ABB RobotStudio station: YuMi_Final_10-14-18.rspag

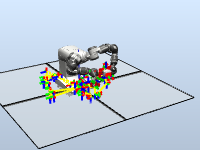
--- station ---
Station YuMi_Capstone_Final (saved by RobotStudio 6.7.7936.1011)
Controller Yumi_LF_Offline
  mechanical unit ROB_R: IRB14000_0.5_0.5_R, 6 joints, base frame (0, 0, 0) mm
  mechanical unit ROB_R_7: IRB14000_0.5_0.5_R, 1 joints, base frame (0, 0, 0) mm
  mechanical unit ROB_L: IRB14000_0.5_0.5_L, 6 joints, base frame (0, 0, 0) mm
  mechanical unit ROB_L_7: IRB14000_0.5_0.5_L, 1 joints, base frame (0, 0, 0) mm
Layout (positions relative to the parent item):
  - Smart_Gripper_Servo_One_Vacuum_Camera_Fingers [mechanism, from Tools\ABB_Smart_Gripper_Servo_One_Vacuum_Camera_Fingers.rslib] at (391.27, -12.04, 287.62) mm, rotated rx 179.56 ry 0.03 rz 94.75 deg; joint values [0.025] (rad or m)
  - Smart_Gripper_Servo_One_Vacuum_Camera_Fingers_2 [mechanism, from Tools\ABB_Smart_Gripper_Servo_One_Vacuum_Camera_Fingers.rslib] at (282.29, 267.76, 240.04) mm, rotated rx -93.42 ry -87.31 rz -179.37 deg; joint values [0.025] (rad or m)
  - IRB14000_0.5_0.5_2 [mechanism, from Robots\IRB14000_0.5_0.5__01.rslib] at (0, 0, 0) mm
  - IRB14000_0.5_0.5_R [mechanism, from Robots\IRB14000_0.5_0.5__01.rslib] at (0, 0, 0) mm; joint values [1.4938, -0.7266, -1.3651, 0.7569, 4.3395, 1.3243, -3.2623] (rad or m)
  - IRB14000_0.5_0.5_L [mechanism, from Robots\IRB14000_0.5_0.5__01.rslib] at (0, 0, 0) mm; joint values [-0.6453, -1.1889, 1.5214, 0.5648, 0.0097, 1.2191, -0.4517] (rad or m)
Attachment: Smart_Gripper_Servo_One_Vacuum_Camera_Fingers is attached to IRB14000_0.5_0.5_R / Link7
Attachment: Smart_Gripper_Servo_One_Vacuum_Camera_Fingers_2 is attached to IRB14000_0.5_0.5_L / Link7
Targets, tools, work objects and paths stored in the station and not in the controller backup, written as RAPID:
! task T_ROB_R
MODULE MainModule
  VAR syncident sync1;
  VAR syncident sync2;
  VAR syncident sync3;
  VAR syncident sync4;
  VAR syncident sync5;
  VAR syncident sync6;
  VAR syncident sync7;
  VAR syncident sync8;
  VAR syncident sync9;
  VAR syncident sync10;
  VAR syncident sync11;
  VAR syncident sync12;
  VAR syncident sync13;
  VAR syncident sync14;
  VAR syncident sync15;
  VAR syncident sync16;
  VAR syncident sync17;
ENDMODULE

! task T_ROB_R
MODULE CalibData
  PERS tooldata Servo:=[TRUE,[[0,0,114.2],[1,0,0,0]],[0.24,[8.2,12.5,48.1],[1,0,0,0],0.00022,0.00024,0.00009]];
  PERS tooldata VaccumOne:=[TRUE,[[56,18.5,37.5],[0.707106781,0,0.707106781,0]],[0.24,[8.2,12.5,48.1],[1,0,0,0],0.00022,0.00024,0.00009]];
  PERS tooldata Camera:=[TRUE,[[-7.3,28.3,35.1],[0.5,-0.5,0.5,0.5]],[0.24,[8.2,12.5,48.1],[1,0,0,0],0.00022,0.00024,0.00009]];
ENDMODULE

! task T_ROB_L
MODULE MainModule
  VAR syncident sync1;
  VAR syncident sync2;
  VAR syncident sync3;
  VAR syncident sync4;
  VAR syncident sync5;
  VAR syncident sync6;
  VAR syncident sync7;
  VAR syncident sync8;
  VAR syncident sync9;
  VAR syncident sync10;
  VAR syncident sync11;
  VAR syncident sync12;
  VAR syncident sync13;
  VAR syncident sync14;
  VAR syncident sync15;
  VAR syncident sync16;
  VAR syncident sync17;
ENDMODULE

! task T_ROB_L
MODULE CalibData
  PERS tooldata Servo:=[TRUE,[[0,0,114.2],[1,0,0,0]],[0.24,[8.2,12.5,48.1],[1,0,0,0],0.00022,0.00024,0.00009]];
  PERS tooldata VaccumOne:=[TRUE,[[56,18.5,37.5],[0.707106781,0,0.707106781,0]],[0.24,[8.2,12.5,48.1],[1,0,0,0],0.00022,0.00024,0.00009]];
  PERS tooldata Camera:=[TRUE,[[-7.3,28.3,35.1],[0.5,-0.5,0.5,0.5]],[0.24,[8.2,12.5,48.1],[1,0,0,0],0.00022,0.00024,0.00009]];
ENDMODULE

! task T_ROB_R
MODULE CalibData
  PERS tooldata Servo:=[TRUE,[[0,0,114.2],[1,0,0,0]],[0.24,[8.2,12.5,48.1],[1,0,0,0],0.00022,0.00024,0.00009]];
  PERS tooldata VaccumOne:=[TRUE,[[56,18.5,37.5],[0.707106781,0,0.707106781,0]],[0.24,[8.2,12.5,48.1],[1,0,0,0],0.00022,0.00024,0.00009]];
  PERS tooldata Camera:=[TRUE,[[-7.3,28.3,35.1],[0.5,-0.5,0.5,0.5]],[0.24,[8.2,12.5,48.1],[1,0,0,0],0.00022,0.00024,0.00009]];
ENDMODULE

! task T_ROB_L
MODULE CalibData
  PERS tooldata Servo:=[TRUE,[[0,0,114.2],[1,0,0,0]],[0.24,[8.2,12.5,48.1],[1,0,0,0],0.00022,0.00024,0.00009]];
  PERS tooldata VaccumOne:=[TRUE,[[56,18.5,37.5],[0.707106781,0,0.707106781,0]],[0.24,[8.2,12.5,48.1],[1,0,0,0],0.00022,0.00024,0.00009]];
  PERS tooldata Camera:=[TRUE,[[-7.3,28.3,35.1],[0.5,-0.5,0.5,0.5]],[0.24,[8.2,12.5,48.1],[1,0,0,0],0.00022,0.00024,0.00009]];
ENDMODULE


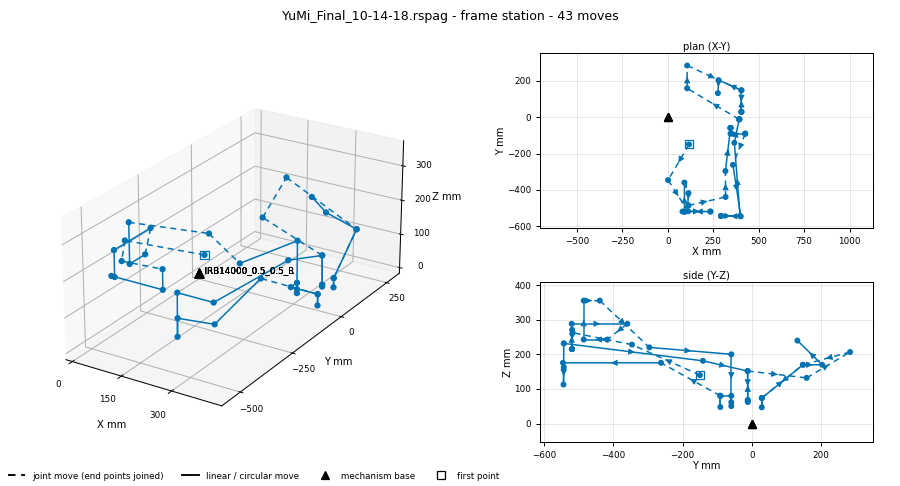
[picture p0: tool path of YuMi_Final_10-14-18.rspag in frame station, 43 of 43 moves have a stored position in this frame; points joined in program order, loops and branches not executed]
--- Backups/Yumi_LF_Offline/RAPID/TASK1/PROGMOD/MainModule.mod ---
MODULE MainModule
    !******************************************************************
    !* Station : YuMi Work Cell
    !******************************************************************
    !* Customer : McMaster University
    !* Project Name : Electronic Screwdriver Assembly
    !*
    !* Robot Model : IRB 14000
    !* Software : RobotWare 6.07
    !*
    !* Authors : Simran Nijjar, Justin Grimm, Samony Riyaz, Amy Hasselman
    !* Company : McMaster University
    !* City/Province : Hamilton, Ontario
    !* Department : W. Booth School of Engineering Practice & Technology
    !* Telephone : N/A
    !*
    !* Program: T_ROB_R
    !* Created : 2018-09-18
    !* Version : 1.0
    !*
    !******************************************************************

    !General Declaration
    PERS tasks task_list{2} := [ ["T_ROB_R"], ["T_ROB_L"] ];
    VAR syncident sync1; !Sync Arm Home Positions
    VAR syncident sync2; !Sync Gripper Open Position
    VAR syncident sync3; !Sync Gripper Close Position
    VAR syncident sync4; !Sync GrommetBin Position1
    VAR syncident sync5; !Sync GrommetBin Position2
    VAR syncident sync6; !Sync GrommetBin Position3
    VAR syncident sync7; !Sync GrommetBin Position4

    !Communication Declaration
    VAR socketdev server;
    VAR socketdev client;
    VAR string message;
    VAR rawbytes data;


	PROC main()
        !Move to Home Position
		MoveJ [[116.737861724,-149.931251033,139.878323961],[0.062653888,-0.842399836,-0.108469979,-0.524090898],[0,0,0,4],[-101.221,9E+09,9E+09,9E+09,9E+09,9E+09]], v1000, z50, tGripper;
		!MoveJ [[110.29,-313.83,302.97],[0.320874,0.00713782,0.947055,0.00865406],[0,1,2,5],[-110.474,9E+09,9E+09,9E+09,9E+09,9E+09]], v1000, z50, tool0;
        WaitSyncTask \InPos, sync1, task_list \TimeOut := 60;

        !Calibrate Grippers
        GripperInitialization;

        !Grippers Initialized Comformation
        g_MoveTo 0;
        WaitRob \InPos;
        WaitSyncTask \InPos, sync2, task_list \TimeOut := 60;

        g_MoveTo 15;
        WaitRob \InPos;
        WaitSyncTask \InPos, sync3, task_list \TimeOut := 60;

        !Move Screwdriver Bin to Correct Position
        MoveJ [[1.625300521,-346.188591473,227.922111416],[0.007707619,0.999903927,-0.000742016,0.011496899],[0,-1,1,4],[-70.2983,9E+09,9E+09,9E+09,9E+09,9E+09]], v1000, z50, tGripper;
        MoveJ [[111.921573894,-517.679338441,262.371959938],[0.007636972,0.999904216,-0.000728005,0.011519802],[0,-1,2,4],[-72.7464,9E+09,9E+09,9E+09,9E+09,9E+09]], v1000, z50, tGripper;
        MoveJ [[234.314486144,-519.240905612,270.651668137],[0.007608269,0.999904877,-0.0005289,0.011492199],[0,-1,2,4],[-162.822,9E+09,9E+09,9E+09,9E+09,9E+09]], v1000, z50, tGripper;
        g_MoveTo 0;
        WaitRob \InPos;
        MoveL [[234.312932861,-519.240747252,215.101630035],[0.00760767,0.999904947,-0.000530615,0.011486499],[0,-1,2,4],[-162.825,9E+09,9E+09,9E+09,9E+09,9E+09]], v1000, z50, tGripper;
        MoveL [[80.782123738,-519.239699323,215.101595493],[0.00760385,0.999905012,-0.00052779,0.0114835],[0,0,1,4],[-162.828,9E+09,9E+09,9E+09,9E+09,9E+09]], v100, z50, tGripper;
        MoveL [[91.392040059,-520.360093654,215.101599575],[0.00760529,0.999905004,-0.000528675,0.0114832],[0,0,1,4],[-162.831,9E+09,9E+09,9E+09,9E+09,9E+09]], v200, z50, tGripper;
        MoveL [[91.399265315,-520.341509224,288.241945811],[0.007536403,0.999904343,-0.000572503,0.011583604],[0,-1,1,4],[-46.5055,9E+09,9E+09,9E+09,9E+09,9E+09]], v200, z50, tGripper;
        WaitRob \InPos;
        MoveL [[91.398688306,-359.668522139,288.241887402],[0.007525373,0.999904448,-0.00057653,0.011581505],[0,-1,2,4],[-46.5056,9E+09,9E+09,9E+09,9E+09,9E+09]], v200, z50, tGripper;
        WaitRob \InPos;
        MoveJ [[113.281646346,-417.364249351,242.672999782],[0.496441086,0.502834087,-0.499757087,0.500946087],[0,1,-1,4],[-119.673,9E+09,9E+09,9E+09,9E+09,9E+09]], v200, z50, tGripper;

        g_MoveTo 9;
        WaitRob \InPos;
        MoveL [[113.281646863,-485.724250766,242.673272807],[0.496441087,0.502833088,-0.499757088,0.500947088],[0,1,0,4],[-119.673,9E+09,9E+09,9E+09,9E+09,9E+09]], v200, z50, tGripper;
        WaitRob \InPos;
        g_GripIn \holdForce :=12;
        MoveL [[113.282188675,-485.724252296,355.154359115],[0.496443089,0.502833091,-0.49975309,0.50094909],[0,2,0,4],[-119.675,9E+09,9E+09,9E+09,9E+09,9E+09]], v200, z50, tGripper;
        MoveJ [[317.912323563,-439.194244895,355.153131276],[0.496442332,0.502837336,-0.499753334,0.500945335],[1,1,-1,4],[-119.678,9E+09,9E+09,9E+09,9E+09,9E+09]], v200, z50, tGripper;
        MoveJ [[317.022439031,-296.105779981,220.044708012],[0.0188621,-0.709563985,0.704158986,0.0179804],[1,3,-1,4],[-119.677,9E+09,9E+09,9E+09,9E+09,9E+09]], v200, z50, tGripper;
        MoveL [[344.96,-59.21,200.05],[0.00733667,-0.709769,0.704368,0.00639342],[1,3,0,4],[157.039,9E+09,9E+09,9E+09,9E+09,9E+09]], v200, z50, tGripper;
        WaitSyncTask \InPos, sync4, task_list \TimeOut := 60;
        MoveL [[344.96,-59.21,61.37],[0.00734294,-0.709766,0.70437,0.00639399],[1,3,0,4],[157.041,9E+09,9E+09,9E+09,9E+09,9E+09]], v20, z50, tGripper;
        MoveL [[344.96,-59.21,50.36],[0.00734279,-0.709765,0.704371,0.00639592],[1,3,0,4],[157.039,9E+09,9E+09,9E+09,9E+09,9E+09]], v20, z50, tGripper;
        WaitRob \InPos;
        g_MoveTo 6;
        WaitRob \InPos;
        WaitSyncTask \InPos, sync5, task_list \TimeOut := 60;
        WaitSyncTask \InPos, sync6, task_list \TimeOut := 60;
        MoveL [[344.95,-59.21,80.07],[0.0073388,-0.709769,0.704367,0.00639981],[1,3,0,4],[157.039,9E+09,9E+09,9E+09,9E+09,9E+09]], v20, z50, tGripper;
        MoveL [[344.95,-90.89,80.07],[0.00733899,-0.70977,0.704366,0.00640178],[1,3,0,4],[157.038,9E+09,9E+09,9E+09,9E+09,9E+09]], v20, z50, tGripper;
        WaitSyncTask \InPos, sync7, task_list \TimeOut := 60;
        MoveL [[425.74,-90.89,80.07],[0.00733914,-0.709769,0.704367,0.00640155],[1,3,0,4],[157.038,9E+09,9E+09,9E+09,9E+09,9E+09]], v20, z50, tGripper;
        MoveL [[425.74,-90.89,47.66],[0.00734079,-0.709768,0.704368,0.00640208],[1,3,0,4],[157.038,9E+09,9E+09,9E+09,9E+09,9E+09]], v20, z50, tGripper;
        WaitRob \InPos;
        g_MoveTo 12;
        WaitRob \InPos;
        MoveL [[425.74,-90.89,80.07],[0.00733914,-0.709769,0.704367,0.00640155],[1,3,0,4],[157.038,9E+09,9E+09,9E+09,9E+09,9E+09]], v20, z50, tGripper;
        MoveJ [[358.12,-262.41,175.42],[0.00734778,-0.709763,0.704373,0.00641492],[0,3,-1,4],[157.036,9E+09,9E+09,9E+09,9E+09,9E+09]], v200, z50, tGripper;
        MoveL [[401.48,-545.66,175.40],[0.00980935,-0.999797,0.0175768,-0.000449508],[1,3,-2,4],[-152.759,9E+09,9E+09,9E+09,9E+09,9E+09]], v200, z50, tGripper;
        MoveL [[292.66,-543.24,162.68],[0.00981674,-0.999797,0.0175764,-0.000446634],[0,3,-2,4],[-152.763,9E+09,9E+09,9E+09,9E+09,9E+09]], v20, z50, tGripper;
        MoveL [[292.39,-544.14,112.56],[0.00982093,-0.999936,-0.00555262,-0.000675012],[0,3,-2,4],[-152.771,9E+09,9E+09,9E+09,9E+09,9E+09]], v20, z50, tGripper;
        WaitRob \InPos;
        g_MoveTo 6;
        WaitRob \InPos;
        g_GripIn \holdForce := 12;
        WaitRob \InPos;
        MoveL [[292.66,-543.25,231.50],[0.00981188,-0.999797,0.0175706,-0.000448127],[0,3,-2,4],[-152.762,9E+09,9E+09,9E+09,9E+09,9E+09]], v20, z50, tGripper;
        MoveL [[397.32,-543.24,231.50],[0.00980798,-0.999797,0.0175712,-0.000449308],[1,3,-2,4],[-152.763,9E+09,9E+09,9E+09,9E+09,9E+09]], v20, z50, tGripper;
        MoveL [[366.17,-140.98,181.13],[0.00267605,0.705528,0.708672,0.00274474],[1,3,-2,4],[166.603,9E+09,9E+09,9E+09,9E+09,9E+09]], v200, z50, tGripper;
        MoveL [[392.31,-12.03,151.62],[0.00277692,0.677184,0.735803,0.00262845],[1,3,-2,4],[166.306,9E+09,9E+09,9E+09,9E+09,9E+09]], v200, z50, tGripper;
        MoveL [[393.44,-11.60,67.62],[0.00277557,0.677187,0.735801,0.0026324],[1,3,-2,4],[166.306,9E+09,9E+09,9E+09,9E+09,9E+09]], v20, z50, tGripper;
        MoveL [[393.44,-11.60,62.17],[0.00277571,0.677187,0.735801,0.00263129],[1,3,-2,4],[166.306,9E+09,9E+09,9E+09,9E+09,9E+09]], v10, z50, tGripper;
        WaitRob \InPos;
        g_MoveTo 12;
        WaitRob \InPos;
        MoveL [[393.44,-11.60,67.62],[0.00277557,0.677187,0.735801,0.0026324],[1,3,-2,4],[166.306,9E+09,9E+09,9E+09,9E+09,9E+09]], v20, z50, tGripper;
        MoveL [[392.31,-12.03,151.62],[0.00277692,0.677184,0.735803,0.00262845],[1,3,-2,4],[166.306,9E+09,9E+09,9E+09,9E+09,9E+09]], v200, z50, tGripper;













!        !Create communication
!        SocketCreate server;
!        SocketBind server, "10.0.13.12", 55000;
!        SocketListen server;
!        SocketAccept server, client;

!        !Send message to the client
!        !SocketSend client\Str:="Hello me!";

!        FOR i FROM 1 TO 10 DO
!            SocketSend client\Str:="Hello me!";
!        ENDFOR


!        !Receive a message from the client
!        SocketReceive client, \RawData:=data;
!        UnpackRawBytes data,1,message\ASCII:=15;

!        !Close communication
!        SocketClose server;


    ENDPROC




    PROC GripperInitialization()
            !Initialization code
            VAR num GripperState;
            VAR bool GripperCalibrated;

            !Check gripper is powered on and calibrated
            GripperState:=g_GetState();
            TPWrite ": Gripper State: "\Num:=GripperState;
            GripperCalibrated:=g_IsCalibrated();

            IF (Not GripperCalibrated) THEN
                g_Init\Calibrate;
            ENDIF

            RETURN;

        ERROR
            IF (ERRNO=ERR_NORUNUNIT) THEN TPWrite " Gripper not powered on.";
                EXIT;
            ENDIF
            TPWrite " Init. - Unhandled Error. #"\Num:=ERRNO;
            EXIT;
    ENDPROC





ENDMODULE

--- Backups/Yumi_LF_Offline/RAPID/TASK1/SYSMOD/LINKEDM.sys ---
%%%
  VERSION:1
  LANGUAGE:ENGLISH
%%%

MODULE LINKEDM (SYSMODULE)

! FOLLOWER
!     Name of electronically linked follower axis used by operator at teach pendent.
      PERS string l_f_axis_name{5}       :=  ["",  "", "", "", ""];

!     Name of the mechanical unit for follower axis.
      PERS string l_f_mecunt_n{5}  :=  ["", "", "", "", ""];

!     Linked follower axis number in the mechanical unit (first axis in mech. unit is number 1).
      PERS num l_f_axis_no{5}      :=  [0,          0,   0,  0,  0];

! MASTER
!     Name of the mechanical unit for linked master axis.
      PERS string l_m_mecunt_n{5} :=  ["", "", "", "", ""];

!     Linked master axis number in the mechanical unit (first axis in mech. unit is number 1).
!     See axis number table in documentation for different master mechanical units.
      PERS num l_m_axis_no{5}     :=  [0,  0,  0,  0,  0];

! POSITION OFFSET
!     The increase of the allowed offset position between the master and follower
!     positions, used when starting AUTO mode. As soon as the offset is decreased
!     the old configurated parameter is used.
!     Example: 3 => the configurated value of allowed offset is increased 3 times.
      PERS num offset_ratio{5}       :=  [10,  10,   10,  10,  10];

! SPEED RATIO
!     Speed_ratio used in AUTO and JOG modes [ very_slow   slow    normal    fast]
!     Value 1 = max allowed manual speed.
      CONST num speed_ratio {20}      := [0.01, 0.01, 0.01, 0.01, 0.01,
                                          0.05, 0.05, 0.05, 0.05, 0.05,
                                          0.20, 0.20, 0.20, 0.20, 0.20,
                                          1.00, 1.00, 1.00, 1.00, 1.00];

! STEP SIZE
!     Displacement position used in JOG mode for each activation of positive or
!     negative movement.                  [very_short    short   normal   long]
!     Unit degees or meter.
      CONST num displacement {20}     := [0.001, 0.001, 0.001, 0.001, 0.001,
                                          0.005, 0.005, 0.005, 0.005, 0.005,
                                          0.020, 0.020, 0.020, 0.020, 0.020,
                                          0.100, 0.100, 0.100, 0.100, 0.100];


!-------------------------------------------------------------
 PROC Linked_m ()
      Linked_m_exe ;
 ENDPROC
ENDMODULE

--- Backups/Yumi_LF_Offline/RAPID/TASK1/SYSMOD/YuMiLib_Params_R.sys ---
MODULE YuMiLib_Params_R(SYSMODULE)
    !***************************************************************************
    !*                              Common parameters                          *
    !***************************************************************************
    CONST loaddata ld_YuMiGripper_S:=[0.230,[8.2,11.7,52.0],[1,0,0,0],0.00021,0.00024,0.00009];
    CONST loaddata ld_YuMiGripper_S_V1:=[0.248,[8.6,11.7,52.7],[1,0,0,0],0.00021,0.00024,0.00009];
    CONST loaddata ld_YuMiGripper_S_V1_V2:=[0.280,[7.1,11.9,47.3],[1,0,0,0],0.00025,0.00029,0.00012];
    CONST loaddata ld_YuMiGripper_S_C:=[0.244,[7.5,11.8,52.7],[1,0,0,0],0.00021,0.00023,0.00008];
    CONST loaddata ld_YuMiGripper_S_C_V1:=[0.262,[7.8,11.9,50.7],[1,0,0,0],0.00022,0.00024,0.00009];

    !***************************************************************************
    ! Predefined tools for different configurations of the Standard Smart Gripper
    !***************************************************************************
    TASK PERS tooldata tHandCamera:=[TRUE,[[-7.79332,26.2553,35.637],[0.507106,-0.492819,-0.512337,-0.487323]],[0.262,[7.8,11.9,50.7],[1,0,0,0],0.00022,0.00024,0.00009]];
    TASK PERS tooldata tGripper:=[TRUE,[[0,0,136],[1,0,0,0]],[0.23,[8.2,11.7,52],[1,0,0,0],0.00021,0.00024,0.00009]];
    TASK PERS tooldata tVacuum1:=[TRUE,[[63.5,18.5,37.5],[0.707106781,0,0.707106781,0]],[0.248,[8.6,11.7,52.7],[1,0,0,0],0.00021,0.00024,0.00009]];
    TASK PERS tooldata tVacuum2:=[TRUE,[[-63.5,18.5,37.5],[0.707106781,0,-0.707106781,0]],[0.28,[7.1,11.9,47.3],[1,0,0,0],0.00025,0.00029,0.00012]];

    !***************************************************************************
    !*                         Task specific paramters                         *
    !***************************************************************************

    TASK PERS wobjdata WObj_FollowRobL:=[FALSE,FALSE,"ROB_L",[[0,0,0],[1,0,0,0]],[[0,0,0],[1,0,0,0]]];
    TASK PERS wobjdata WObj_Vision:=[FALSE,TRUE,"",[[401.591,32.4092,0],[0.424655,-0.000000122,-0.000000191,0.905355]],[[0,0,0],[1,0,0,0]]];

    !**************************************************************************
    !*                                Speeddata                               *
    !**************************************************************************
    CONST speeddata vSlow:=[100,50,5000,1000];
    CONST speeddata vMedium:=[300,150,5000,1000];
    CONST speeddata vFast:=v1000;

ENDMODULE

--- Backups/Yumi_LF_Offline/RAPID/TASK2/PROGMOD/MainModule.mod ---
MODULE MainModule
    !******************************************************************
    !* Station : YuMi Work Cell
    !******************************************************************
    !* Customer : McMaster University
    !* Project Name : Electronic Screwdriver Assembly
    !*
    !* Robot Model : IRB 14000
    !* Software : RobotWare 6.07
    !*
    !* Authors : Simran Nijjar, Justin Grimm, Samony Riyaz, Amy Hasselman
    !* Company : McMaster University
    !* City/Province : Hamilton, Ontario
    !* Department : W. Booth School of Engineering Practice & Technology
    !* Telephone : N/A
    !*
    !* Program: T_ROB_L
    !* Created : 2018-09-18
    !* Version : 1.0
    !*
    !******************************************************************

    !General Declaration
    PERS tasks task_list{2} := [ ["T_ROB_R"], ["T_ROB_L"] ];
    VAR syncident sync1; !Sync Arm Home Positions
    VAR syncident sync2; !Sync Gripper Open Position
    VAR syncident sync3; !Sync Gripper Close Position
    VAR syncident sync4; !Sync GrommetBin Position1
    VAR syncident sync5; !Sync GrommetBin Position2
    VAR syncident sync6; !Sync GrommetBin Position3
    VAR syncident sync7; !Sync GrommetBin Position4

    !Communication Declaration
    VAR socketdev server;
    VAR socketdev client;
    VAR string message;
    VAR rawbytes data;


    PROC main()
		MoveJ [[106.445211471,158.554553337,131.92293514],[0.04782649,0.851736822,-0.124160974,0.506794894],[0,0,0,4],[101.293,9E+09,9E+09,9E+09,9E+09,9E+09]], v1000, z50, tGripper;
		!MoveJ [[97.79,299.03,304.48],[0.0114881,-0.942459,0.0541276,-0.329712],[0,-2,-2,4],[108.747,9E+09,9E+09,9E+09,9E+09,9E+09]], v1000, z50, tool0;
        WaitSyncTask \InPos, sync1, task_list \TimeOut := 60;

        !Calibrate Grippers
        GripperInitialization;

        !Grippers Initialized Comformation
        g_MoveTo 0;
        WaitRob \InPos;
        WaitSyncTask \InPos, sync2, task_list \TimeOut := 60;

        g_MoveTo 15;
        WaitRob \InPos;
        WaitSyncTask \InPos, sync3, task_list \TimeOut := 60;

        !Remove Grommet from Right Screwdriver Shell
        WaitSyncTask \InPos, sync4, task_list \TimeOut := 60;
        MoveJ [[106.46,283.94,206.53],[0.0478122,0.85173,-0.124169,0.506805],[0,0,0,4],[101.295,9E+09,9E+09,9E+09,9E+09,9E+09]], v200, z50, tGripper;
        MoveJ [[404.90,147.80,169.77],[0.009872,-0.723527,-0.690004,0.0174687],[-1,1,0,4],[-169.944,9E+09,9E+09,9E+09,9E+09,9E+09]], v200, z50, tGripper;
        WaitSyncTask \InPos, sync5, task_list \TimeOut := 60;
        MoveL [[404.90,28.94,73.67],[0.0098782,-0.723515,-0.690017,0.0174677],[-1,2,0,4],[146.542,9E+09,9E+09,9E+09,9E+09,9E+09]], v200, z50, tGripper;
        MoveL [[404.90,28.94,46.77],[0.0098791,-0.723519,-0.690013,0.017455],[-1,2,0,4],[146.542,9E+09,9E+09,9E+09,9E+09,9E+09]], v20, z50, tGripper;
        WaitSyncTask \InPos, sync6, task_list \TimeOut := 60;
        WaitSyncTask \InPos, sync7, task_list \TimeOut := 60;
        MoveL [[404.90,28.94,73.67],[0.0098782,-0.723515,-0.690017,0.0174677],[-1,2,0,4],[146.542,9E+09,9E+09,9E+09,9E+09,9E+09]], v200, z50, tGripper;
        MoveJ [[404.90,147.80,169.77],[0.009872,-0.723527,-0.690004,0.0174687],[-1,1,0,4],[-169.944,9E+09,9E+09,9E+09,9E+09,9E+09]], v200, z50, tGripper;
        MoveL [[279.71,203.37,169.78],[0.0174576,0.685927,-0.727395,-0.00975931],[0,1,-2,4],[-169.942,9E+09,9E+09,9E+09,9E+09,9E+09]], v200, z50, tGripper;
        WaitRob \InPos;
        MoveL [[275.69,131.92,239.66],[0.499697,0.476231,-0.524027,0.498901],[0,0,0,4],[-175.134,9E+09,9E+09,9E+09,9E+09,9E+09]], v200, z50, tGripper;
        g_MoveTo 12;






!        !Vacuum Controls
!        VacuumTool_ON;
!        WaitTime(10);
!        VacuumTool_OFF;




!        !Create communication
!        SocketCreate server;
!        SocketBind server, "10.0.13.12", 55000;
!        SocketListen server;
!        SocketAccept server, client;

!        !Send message to the client
!        !SocketSend client\Str:="Hello me!";

!        FOR i FROM 1 TO 10 DO
!            SocketSend client\Str:="Hello me!";
!        ENDFOR


!        !Receive a message from the client
!        SocketReceive client, \RawData:=data;
!        UnpackRawBytes data,1,message\ASCII:=15;

!        !Close communication
!        SocketClose server;
    ENDPROC




    PROC GripperInitialization()
            !Initialization code
            VAR num GripperState;
            VAR bool GripperCalibrated;

            !Check gripper is powered on and calibrated.
            GripperState:=g_GetState();
            TPWrite ": Gripper State: "\Num:=GripperState;
            GripperCalibrated:=g_IsCalibrated();

            IF (Not GripperCalibrated) THEN
                g_Init\Calibrate;
            ENDIF
        RETURN;

        ERROR
            IF (ERRNO=ERR_NORUNUNIT) THEN TPWrite " Gripper not powered on.";
                EXIT;
            ENDIF
            TPWrite " Init. - Unhandled Error. #"\Num:=ERRNO;
            EXIT;
    ENDPROC


    PROC VacuumTool_OFF()
        SetDO Tool_Suction_ON, 0; !Check Logic to confirm that the solenoid valve is in the neutral state before turning off
        SetDO Tool_Suction_OFF, 1;
        WaitTime(0.5);
        SetDO Tool_Suction_OFF, 0;
    ENDPROC


    PROC VacuumTool_ON()
        SetDO Tool_Suction_OFF, 0; !Check Logic to confirm that the solenoid valve is in the neutral state before turning on
        SetDO Tool_Suction_ON, 1;
        WaitTime(0.5);
        SetDO Tool_Suction_ON, 0;
    ENDPROC


ENDMODULE

--- Backups/Yumi_LF_Offline/RAPID/TASK2/SYSMOD/YuMiLib_Params_L.sys ---
MODULE YuMiLib_Params_L(SYSMODULE)
    !***************************************************************************
    !*                              Common parameters                          *
    !***************************************************************************
    CONST loaddata ld_YuMiGripper_S:=[0.230,[8.2,11.7,52.0],[1,0,0,0],0.00021,0.00024,0.00009];
    CONST loaddata ld_YuMiGripper_S_V1:=[0.248,[8.6,11.7,52.7],[1,0,0,0],0.00021,0.00024,0.00009];
    CONST loaddata ld_YuMiGripper_S_V1_V2:=[0.280,[7.1,11.9,47.3],[1,0,0,0],0.00025,0.00029,0.00012];
    CONST loaddata ld_YuMiGripper_S_C:=[0.244,[7.5,11.8,52.7],[1,0,0,0],0.00021,0.00023,0.00008];
    CONST loaddata ld_YuMiGripper_S_C_V1:=[0.262,[7.8,11.9,50.7],[1,0,0,0],0.00022,0.00024,0.00009];

    !***************************************************************************
    ! Predefined tools for different configurations of the Standard Smart Gripper
    !***************************************************************************
    TASK PERS tooldata tHandCamera:=[TRUE,[[-7.79332,26.2553,35.637],[0.507106,-0.492819,-0.512337,-0.487323]],[0.262,[7.8,11.9,50.7],[1,0,0,0],0.00022,0.00024,0.00009]];
    TASK PERS tooldata tGripper:=[TRUE,[[0,0,136],[1,0,0,0]],[0.23,[8.2,11.7,52],[1,0,0,0],0.00021,0.00024,0.00009]];
    TASK PERS tooldata tVacuum1:=[TRUE,[[63.5,18.5,37.5],[0.707106781,0,0.707106781,0]],[0.248,[8.6,11.7,52.7],[1,0,0,0],0.00021,0.00024,0.00009]];
    TASK PERS tooldata tVacuum2:=[TRUE,[[-63.5,18.5,37.5],[0.707106781,0,-0.707106781,0]],[0.280,[7.1,11.9,47.3],[1,0,0,0],0.00025,0.00029,0.00012]];

    !***************************************************************************
    !*                         Task specific paramters                         *
    !***************************************************************************

    TASK PERS wobjdata WObj_FollowRobR:=[FALSE,FALSE,"ROB_R",[[0,0,0],[1,0,0,0]],[[0,0,0],[1,0,0,0]]];
    TASK PERS wobjdata WObj_Vision:=[FALSE,TRUE,"",[[401.591,32.4092,0],[0.424655,-1.21554E-07,-1.90773E-07,0.905355]],[[0,0,0],[1,0,0,0]]];

    !**************************************************************************
    !*                                Speeddata                               *
    !**************************************************************************

    CONST speeddata vSlow:=[100,50,5000,1000];
    CONST speeddata vMedium:=[300,150,5000,1000];
    CONST speeddata vFast:=v1000;
ENDMODULE

--- Backups/Yumi_LF_Offline/SYSPAR/EIO.cfg ---
EIO:CFG_1.0:6:1::
#
SYSSIG_IN:

      -Signal "Collision_Avoidance" -Action "CollAvoidance"
#
INDUSTRIAL_NETWORK:

      -Name "EtherNetIP" -Connection "Private Network" -Label "EtherNet/IP"

      -Name "DeviceNet" -Label "DeviceNet Master/Slave Network" -Address "2"

      -Name "EtherNetIP_Anybus" -Label "EtherNet/IP Anybus Network"\
      -Address "0.0.0.0" -SubnetMask "255.255.255.0" -Gateway "0.0.0.0"
#
EIO_CROSS:

      -Name "Cross_Signal_Lamp" -Res "Signal_Lamp" -Act1 "DRV1BRAKE"
#
EIO_SIGNAL_SAFELEVEL:

      -Name "FlangePowerSafeLevel" -ActionWhenStartup "Last"

      -Name "SGcmdSafeLevel" -ActionWhenAccessible "Default"
#
ETHERNETIP_DEVICE:

      -Name "Hand_R" -StateWhenStartup "Deactivated" -VendorName "ABB"\
      -ProductName "EtherNet/IP EIP" -Label "2" -Address "192.168.125.30"\
      -VendorId 75 -ProductCode 1 -OutputAssembly 100 -InputAssembly 101\
      -InputConnectionType "POINT2POINT" -OutputSize 10 -InputSize 10\
      -O2T_RPI 10000 -T2O_RPI 10000 -ConnectionTimeoutMultiplier 2

      -Name "Hand_L" -StateWhenStartup "Deactivated" -VendorName "ABB"\
      -ProductName "EtherNet/IP EIP" -Label "1" -Address "192.168.125.40"\
      -VendorId 75 -ProductCode 1 -OutputAssembly 100 -InputAssembly 101\
      -InputConnectionType "POINT2POINT" -OutputSize 10 -InputSize 10\
      -O2T_RPI 10000 -T2O_RPI 10000 -ConnectionTimeoutMultiplier 2
#
DEVICENET_DEVICE:

      -Name "D652_10" -VendorName "ABB Robotics" -ProductName "24 VDC Unit"\
      -Address 10 -ProductCode 26 -DeviceType 7 -ConnectionType "COS"\
      -OutputSize 2 -InputSize 2
#
DEVICENET_INTERNAL_DEVICE:

      -Name "DN_Internal_Device" -VendorName "ABB Robotics"\
      -ProductName "DeviceNet Internal Slave Device"
#
ETHERNETIP_INTERNAL_DEVICE:

      -Name "EN_Internal_Device" -VendorName "ABB Robotics"\
      -ProductName "EtherNet/IP Internal Adapter Device"
#
ETHERNETIP_INTERNAL_ANYBUS_DEVICE:

      -Name "EN_Internal_Anybus" -VendorName "ABB Robotics"\
      -ProductName "EtherNet/IP Internal Anybus Adapter Device"
#
EIO_SIGNAL:

      -Name "custom_DI_0" -SignalType "DI" -Device "D652_10" -DeviceMap "0"

      -Name "custom_DI_1" -SignalType "DI" -Device "D652_10" -DeviceMap "1"

      -Name "custom_DI_2" -SignalType "DI" -Device "D652_10" -DeviceMap "2"

      -Name "custom_DI_3" -SignalType "DI" -Device "D652_10" -DeviceMap "3"

      -Name "custom_DI_4" -SignalType "DI" -Device "D652_10" -DeviceMap "4"

      -Name "custom_DI_5" -SignalType "DI" -Device "D652_10" -DeviceMap "5"

      -Name "custom_DI_6" -SignalType "DI" -Device "D652_10" -DeviceMap "6"

      -Name "custom_DI_7" -SignalType "DI" -Device "D652_10" -DeviceMap "7"

      -Name "Tool_Suction_OFF" -SignalType "DO" -Device "D652_10"\
      -Label "custom_DO_0" -DeviceMap "0"

      -Name "Tool_Suction_ON" -SignalType "DO" -Device "D652_10"\
      -Label "custom_DO_1" -DeviceMap "1"

      -Name "custom_DO_2" -SignalType "DO" -Device "D652_10" -DeviceMap "2"

      -Name "custom_DO_3" -SignalType "DO" -Device "D652_10" -DeviceMap "3"

      -Name "custom_DO_4" -SignalType "DO" -Device "D652_10" -DeviceMap "4"

      -Name "custom_DO_5" -SignalType "DO" -Device "D652_10" -DeviceMap "5"

      -Name "custom_DO_6" -SignalType "DO" -Device "D652_10" -DeviceMap "6"

      -Name "custom_DO_7" -SignalType "DO" -Device "D652_10" -DeviceMap "7"

      -Name "hall_sensor_joint_1" -SignalType "DI" -Device "D652_10"\
      -DeviceMap "8"

      -Name "hall_sensor_joint_2" -SignalType "DI" -Device "D652_10"\
      -DeviceMap "9"

      -Name "hall_sensor_joint_3" -SignalType "DI" -Device "D652_10"\
      -DeviceMap "11"

      -Name "hall_sensor_joint_4" -SignalType "DI" -Device "D652_10"\
      -DeviceMap "12"

      -Name "hall_sensor_joint_5" -SignalType "DI" -Device "D652_10"\
      -DeviceMap "13"

      -Name "hall_sensor_joint_6" -SignalType "DI" -Device "D652_10"\
      -DeviceMap "14"

      -Name "hall_sensor_joint_7" -SignalType "DI" -Device "D652_10"\
      -DeviceMap "10"

      -Name "hall_sensor_24V_ROB_R" -SignalType "DO" -Device "D652_10"\
      -DeviceMap "8"

      -Name "hall_sensor_24V_ROB_L" -SignalType "DO" -Device "D652_10"\
      -DeviceMap "9"

      -Name "flange_24V_ROB_R" -SignalType "DO" -Device "D652_10"\
      -DeviceMap "10" -SafeLevel "FlangePowerSafeLevel"

      -Name "flange_24V_ROB_L" -SignalType "DO" -Device "D652_10"\
      -DeviceMap "11" -SafeLevel "FlangePowerSafeLevel"

      -Name "Signal_Lamp" -SignalType "DO" -Device "D652_10" -DeviceMap "12"

      -Name "Collision_Avoidance" -SignalType "DO" -Access "All" -Default 1

      -Name "hand_CmdGripper_R" -SignalType "GO" -Device "Hand_R"\
      -Label "Hand Command Right" -DeviceMap "0-4" -Category "HandRight"\
      -Access "All" -SafeLevel "SGcmdSafeLevel"

      -Name "hand_CmdClearErr_R" -SignalType "DO" -Device "Hand_R"\
      -Label "Clear Error Right" -DeviceMap "7" -Category "HandRight"\
      -Access "All"

      -Name "hand_MaxPosition_R" -SignalType "GO" -Device "Hand_R"\
      -Label "Max Position Right" -DeviceMap "8-15" -Category "HandRight"\
      -Access "All" -Default 100

      -Name "hand_MinPosition_R" -SignalType "GO" -Device "Hand_R"\
      -Label "Min Position Right" -DeviceMap "16-23" -Category "HandRight"\
      -Access "All" -Default 50

      -Name "hand_MaxSpeed_R" -SignalType "GO" -Device "Hand_R"\
      -Label "Max Speed Right" -DeviceMap "24-31" -Category "HandRight"\
      -Access "All" -Default 200

      -Name "hand_HoldForce_R" -SignalType "GO" -Device "Hand_R"\
      -Label "Hold Force Right" -DeviceMap "40-47" -Category "HandRight"\
      -Access "All" -Default 120

      -Name "hand_CmdVacuum1_R" -SignalType "DO" -Device "Hand_R"\
      -Label "Vacuum 1 Right" -DeviceMap "48" -Category "HandRight"\
      -Access "All"

      -Name "hand_CmdVacuum2_R" -SignalType "DO" -Device "Hand_R"\
      -Label "Vacuum 2 Right" -DeviceMap "49" -Category "HandRight"\
      -Access "All"

      -Name "hand_CmdBlowoff1_R" -SignalType "DO" -Device "Hand_R"\
      -Label "BlowOff 1 Right" -DeviceMap "50" -Category "HandRight"\
      -Access "All"

      -Name "hand_CmdBlowoff2_R" -SignalType "DO" -Device "Hand_R"\
      -Label "BlowOff 2 Right" -DeviceMap "51" -Category "HandRight"\
      -Access "All"

      -Name "hand_SysState_R" -SignalType "GI" -Device "Hand_R"\
      -Label "Finger State Right" -DeviceMap "0-4" -Category "HandRight"\
      -Access "All"

      -Name "hand_SysError_R" -SignalType "GI" -Device "Hand_R"\
      -Label "Finger Error Right" -DeviceMap "32-39" -Category "HandRight"\
      -Access "All"

      -Name "hand_StatusCalibrated_R" -SignalType "DI" -Device "Hand_R"\
      -Label "Calibrated Right" -DeviceMap "5" -Category "HandRight"\
      -Access "All"

      -Name "hand_ActualPosition_R" -SignalType "GI" -Device "Hand_R"\
      -Label "Actual Position Right" -DeviceMap "8-15" -Category "HandRight"\
      -Access "All"

      -Name "hand_ActualSpeed_R" -SignalType "GI" -Device "Hand_R"\
      -Label "Actual Speed Right" -DeviceMap "16-23" -Category "HandRight"\
      -Access "All"

      -Name "hand_StatusCamLinked_R" -SignalType "DI" -Device "Hand_R"\
      -Label "Camera Connection Right" -DeviceMap "40" -Category "HandRight"\
      -Access "All"

      -Name "hand_SoftwareVersion_R" -SignalType "GI" -Device "Hand_R"\
      -Label "Software Version Right" -DeviceMap "41-47" -Category "HandRight"\
      -Access "All"

      -Name "hand_StatusVacuum1_R" -SignalType "DI" -Device "Hand_R"\
      -Label "Vacuum 1 Right Status" -DeviceMap "48" -Category "HandRight"\
      -Access "All"

      -Name "hand_StatusVacuum2_R" -SignalType "DI" -Device "Hand_R"\
      -Label "Vacuum 1 Right Status" -DeviceMap "49" -Category "HandRight"\
      -Access "All"

      -Name "hand_StatusBlowoff1_R" -SignalType "DI" -Device "Hand_R"\
      -Label "SuncTool 1 Right Status" -DeviceMap "50" -Category "HandRight"\
      -Access "All"

      -Name "hand_StatusBlowoff2_R" -SignalType "DI" -Device "Hand_R"\
      -Label "SuncTool 1 Right Status" -DeviceMap "51" -Category "HandRight"\
      -Access "All"

      -Name "hand_ActualPressure1_R" -SignalType "GI" -Device "Hand_R"\
      -Label "Vacuum pressure1 Right" -DeviceMap "64-71" -Category "HandRight"\
      -Access "All"

      -Name "hand_ActualPressure2_R" -SignalType "GI" -Device "Hand_R"\
      -Label "Vacuum pressure2 Right" -DeviceMap "72-79" -Category "HandRight"\
      -Access "All"

      -Name "hand_SecurityKey_R" -SignalType "GO" -Device "Hand_R"\
      -Label "Security key right" -DeviceMap "64-71" -Category "HandRight"\
      -Access "All"

      -Name "hand_TftPFtpMode_R" -SignalType "DI" -Device "Hand_R"\
      -Label "Hand firmware update mode" -DeviceMap "7" -Category "HandRight"\
      -Access "All"

      -Name "hand_CmdGripper_L" -SignalType "GO" -Device "Hand_L"\
      -Label "Hand Command Left" -DeviceMap "0-4" -Category "HandLeft"\
      -Access "All" -SafeLevel "SGcmdSafeLevel"

      -Name "hand_CmdClearErr_L" -SignalType "DO" -Device "Hand_L"\
      -Label "Clear Error Left" -DeviceMap "7" -Category "HandLeft"\
      -Access "All"

      -Name "hand_MaxPosition_L" -SignalType "GO" -Device "Hand_L"\
      -Label "Max Position Left" -DeviceMap "8-15" -Category "HandLeft"\
      -Access "All" -Default 100

      -Name "hand_MinPosition_L" -SignalType "GO" -Device "Hand_L"\
      -Label "Min Position Left" -DeviceMap "16-23" -Category "HandLeft"\
      -Access "All" -Default 50

      -Name "hand_MaxSpeed_L" -SignalType "GO" -Device "Hand_L"\
      -Label "Max Speed Left" -DeviceMap "24-31" -Category "HandLeft"\
      -Access "All" -Default 200

      -Name "hand_HoldForce_L" -SignalType "GO" -Device "Hand_L"\
      -Label "Hold Force Left" -DeviceMap "40-47" -Category "HandLeft"\
      -Access "All" -Default 120

      -Name "hand_CmdVacuum1_L" -SignalType "DO" -Device "Hand_L"\
      -Label "Vacuum 1 Left" -DeviceMap "48" -Category "HandLeft" -Access "All"

      -Name "hand_CmdVacuum2_L" -SignalType "DO" -Device "Hand_L"\
      -Label "Vacuum 2 Left" -DeviceMap "49" -Category "HandLeft" -Access "All"

      -Name "hand_CmdBlowoff1_L" -SignalType "DO" -Device "Hand_L"\
      -Label "BlowOff 1 Left" -DeviceMap "50" -Category "HandLeft" -Access "All"

      -Name "hand_CmdBlowoff2_L" -SignalType "DO" -Device "Hand_L"\
      -Label "BlowOff 2 Left" -DeviceMap "51" -Category "HandLeft" -Access "All"

      -Name "hand_SysState_L" -SignalType "GI" -Device "Hand_L"\
      -Label "Finger State Left" -DeviceMap "0-4" -Category "HandLeft"\
      -Access "All"

      -Name "hand_SysError_L" -SignalType "GI" -Device "Hand_L"\
      -Label "Finger Error Left" -DeviceMap "32-39" -Category "HandLeft"\
      -Access "All"

      -Name "hand_StatusCalibrated_L" -SignalType "DI" -Device "Hand_L"\
      -Label "Calibrated Left" -DeviceMap "5" -Category "HandLeft" -Access "All"

      -Name "hand_ActualPosition_L" -SignalType "GI" -Device "Hand_L"\
      -Label "Actual Position Left" -DeviceMap "8-15" -Category "HandLeft"\
      -Access "All"

      -Name "hand_ActualSpeed_L" -SignalType "GI" -Device "Hand_L"\
      -Label "Actual Speed Left" -DeviceMap "16-23" -Category "HandLeft"\
      -Access "All"

      -Name "hand_StatusCamLinked_L" -SignalType "DI" -Device "Hand_L"\
      -Label "Camera Connection Left" -DeviceMap "40" -Category "HandLeft"\
      -Access "All"

      -Name "hand_SoftwareVersion_L" -SignalType "GI" -Device "Hand_L"\
      -Label "Software Version Left" -DeviceMap "41-47" -Category "HandLeft"\
      -Access "All"

      -Name "hand_StatusVacuum1_L" -SignalType "DI" -Device "Hand_L"\
      -Label "Vacuum 1 Left Status" -DeviceMap "48" -Category "HandLeft"\
      -Access "All"

      -Name "hand_StatusVacuum2_L" -SignalType "DI" -Device "Hand_L"\
      -Label "Vacuum 1 Left Status" -DeviceMap "49" -Category "HandLeft"\
      -Access "All"

      -Name "hand_StatusBlowoff1_L" -SignalType "DI" -Device "Hand_L"\
      -Label "SuncTool 1 Left Status" -DeviceMap "50" -Category "HandLeft"\
      -Access "All"

      -Name "hand_StatusBlowoff2_L" -SignalType "DI" -Device "Hand_L"\
      -Label "SuncTool 1 Left Status" -DeviceMap "51" -Category "HandLeft"\
      -Access "All"

      -Name "hand_ActualPressure1_L" -SignalType "GI" -Device "Hand_L"\
      -Label "Vacuum pressure1 Left" -DeviceMap "64-71" -Category "HandLeft"\
      -Access "All"

      -Name "hand_ActualPressure2_L" -SignalType "GI" -Device "Hand_L"\
      -Label "Vacuum pressure2 Left" -DeviceMap "72-79" -Category "HandLeft"\
      -Access "All"

      -Name "hand_SecurityKey_L" -SignalType "GO" -Device "Hand_L"\
      -Label "Security key Left" -DeviceMap "64-71" -Category "HandLeft"\
      -Access "All"

      -Name "hand_TftPFtpMode_L" -SignalType "DI" -Device "Hand_L"\
      -Label "Hand firmware update mode" -DeviceMap "7" -Category "HandLeft"\
      -Access "All"
